% RSLogix 500 project water_filtration_system.RSS, saved by version 8.30.00.16 %
PROJECT "UNTITLED"    % processor: Bul.1763 MicroLogix 1100 Series B %

PROGRAM FILES
  LAD 2   12 rungs
  LAD 3 "IO"  13 rungs
  LAD 4 "ALARMS"  18 rungs
  LAD 5 "CTRL"  8 rungs
  LAD 6 "HOA"  23 rungs
  LAD 7 "SIM"  7 rungs
  LAD 8 "MODE"  4 rungs
  LAD 9 "BACKWASH"  16 rungs
  LAD 10 "LEVEL"  5 rungs
  LAD 11 "HOURMETER"  8 rungs
  LAD 12 "REVIEW"  7 rungs

DATA FILES
  O0 OUTPUT  4 elements
  I1 INPUT  6 elements
  S2 STATUS  66 elements
  B3 BINARY  7 elements
  T4 TIMER  15 elements
  C5 COUNTER  1 elements
  R6 CONTROL  1 elements
  N7 INTEGER  13 elements
  F8 FLOAT  12 elements
  B9 DIGITAL IO  1 elements
  N10 ANALOG IO  3 elements

LADDER 2
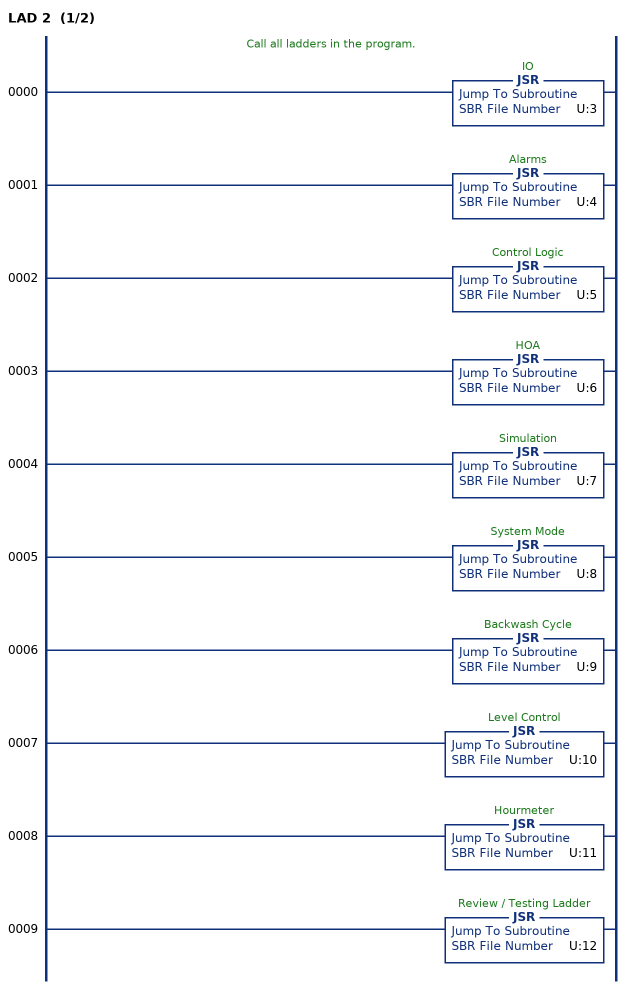
% Rung: 0 %
% Call all ladders in the program. %
SOR JSR U:3 EOR
%   U:3  "IO" %
% Rung: 1 %
SOR JSR U:4 EOR
%   U:4  "Alarms" %
% Rung: 2 %
SOR JSR U:5 EOR
%   U:5  "Control Logic" %
% Rung: 3 %
SOR JSR U:6 EOR
%   U:6  "HOA" %
% Rung: 4 %
SOR JSR U:7 EOR
%   U:7  "Simulation" %
% Rung: 5 %
SOR JSR U:8 EOR
%   U:8  "System Mode" %
% Rung: 6 %
SOR JSR U:9 EOR
%   U:9  "Backwash Cycle" %
% Rung: 7 %
SOR JSR U:10 EOR
%   U:10  "Level Control" %
% Rung: 8 %
SOR JSR U:11 EOR
%   U:11  "Hourmeter" %
% Rung: 9 %
SOR JSR U:12 EOR
%   U:12  "Review / Testing Ladder" %

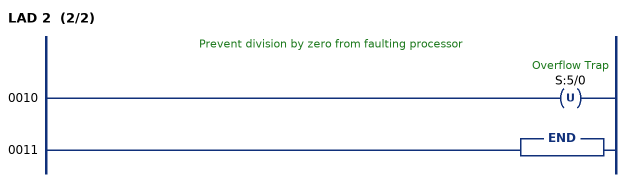
% Rung: 10 %
% Prevent division by zero from faulting processor %
SOR OTU S:5/0 EOR
%   S:5/0  "Overflow Trap" %
% Rung: 11 %
SOR END EOR

LADDER 3 "IO"
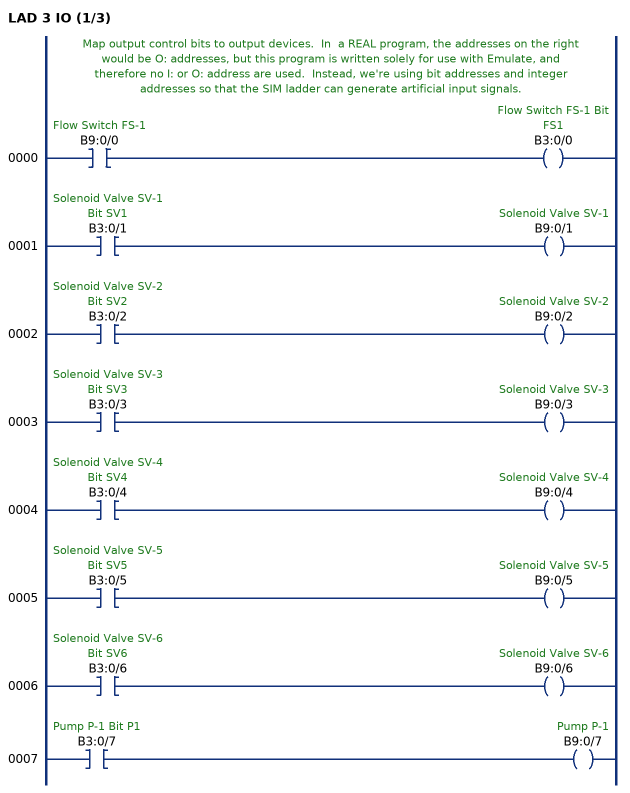
% Rung: 0 %
% Map output control bits to output devices.  In  a REAL program, the addresses on the right would be O: addresses, but this program is written solely for use with Emulate, and therefore no I: or O: address are used.  Instead, we're using bit addresses and integer addresses so that the SIM ladder can generate artificial input signals. %
SOR XIC B9:0/0 OTE B3:0/0 EOR
%   B9:0/0  "Flow Switch FS-1" %
%   B3:0/0  FS1  "Flow Switch FS-1 Bit" %
% Rung: 1 %
SOR XIC B3:0/1 OTE B9:0/1 EOR
%   B3:0/1  SV1  "Solenoid Valve SV-1 Bit" %
%   B9:0/1  "Solenoid Valve SV-1" %
% Rung: 2 %
SOR XIC B3:0/2 OTE B9:0/2 EOR
%   B3:0/2  SV2  "Solenoid Valve SV-2 Bit" %
%   B9:0/2  "Solenoid Valve SV-2" %
% Rung: 3 %
SOR XIC B3:0/3 OTE B9:0/3 EOR
%   B3:0/3  SV3  "Solenoid Valve SV-3 Bit" %
%   B9:0/3  "Solenoid Valve SV-3" %
% Rung: 4 %
SOR XIC B3:0/4 OTE B9:0/4 EOR
%   B3:0/4  SV4  "Solenoid Valve SV-4 Bit" %
%   B9:0/4  "Solenoid Valve SV-4" %
% Rung: 5 %
SOR XIC B3:0/5 OTE B9:0/5 EOR
%   B3:0/5  SV5  "Solenoid Valve SV-5 Bit" %
%   B9:0/5  "Solenoid Valve SV-5" %
% Rung: 6 %
SOR XIC B3:0/6 OTE B9:0/6 EOR
%   B3:0/6  SV6  "Solenoid Valve SV-6 Bit" %
%   B9:0/6  "Solenoid Valve SV-6" %
% Rung: 7 %
SOR XIC B3:0/7 OTE B9:0/7 EOR
%   B3:0/7  P1  "Pump P-1 Bit" %
%   B9:0/7  "Pump P-1" %

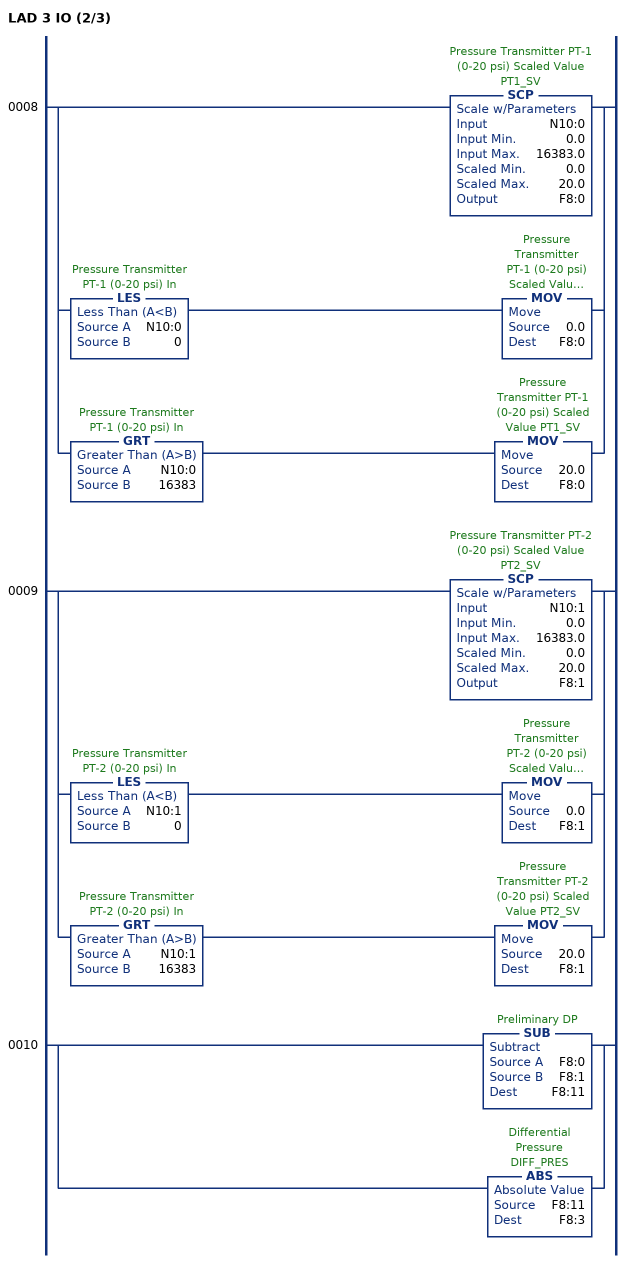
% Rung: 8 %
SOR BST SCP N10:0 0.0 16383.0 0.0 20.0 F8:0 NXB LES N10:0 0 MOV 0.0 F8:0 NXB GRT N10:0 16383 MOV 20.0 F8:0 BND EOR
%   N10:0  "Pressure Transmitter PT-1 (0-20 psi) In" %
%   F8:0  PT1_SV  "Pressure Transmitter PT-1 (0-20 psi) Scaled Value" %
% Rung: 9 %
SOR BST SCP N10:1 0.0 16383.0 0.0 20.0 F8:1 NXB LES N10:1 0 MOV 0.0 F8:1 NXB GRT N10:1 16383 MOV 20.0 F8:1 BND EOR
%   N10:1  "Pressure Transmitter PT-2 (0-20 psi) In" %
%   F8:1  PT2_SV  "Pressure Transmitter PT-2 (0-20 psi) Scaled Value" %
% Rung: 10 %
SOR BST SUB F8:0 F8:1 F8:11 NXB ABS F8:11 F8:3 BND EOR
%   F8:0  PT1_SV  "Pressure Transmitter PT-1 (0-20 psi) Scaled Value" %
%   F8:1  PT2_SV  "Pressure Transmitter PT-2 (0-20 psi) Scaled Value" %
%   F8:11  "Preliminary DP" %
%   F8:3  DIFF_PRES  "Differential Pressure" %

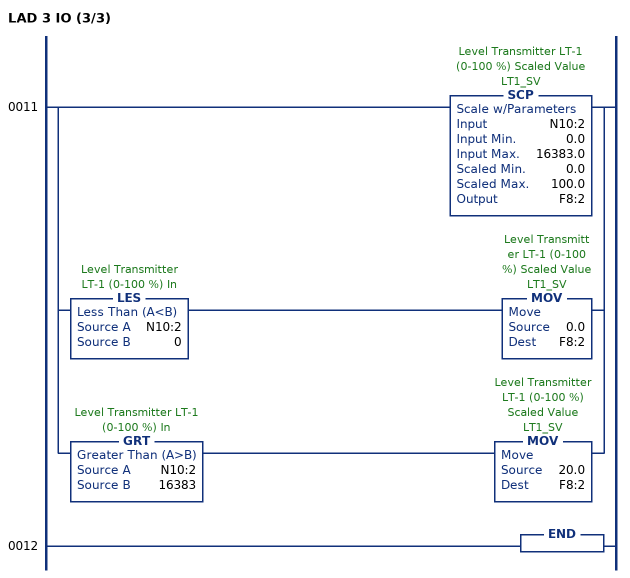
% Rung: 11 %
SOR BST SCP N10:2 0.0 16383.0 0.0 100.0 F8:2 NXB LES N10:2 0 MOV 0.0 F8:2 NXB GRT N10:2 16383 MOV 20.0 F8:2 BND EOR
%   N10:2  "Level Transmitter LT-1 (0-100 %) In" %
%   F8:2  LT1_SV  "Level Transmitter LT-1 (0-100 %) Scaled Value" %
% Rung: 12 %
SOR END EOR

LADDER 4 "ALARMS"
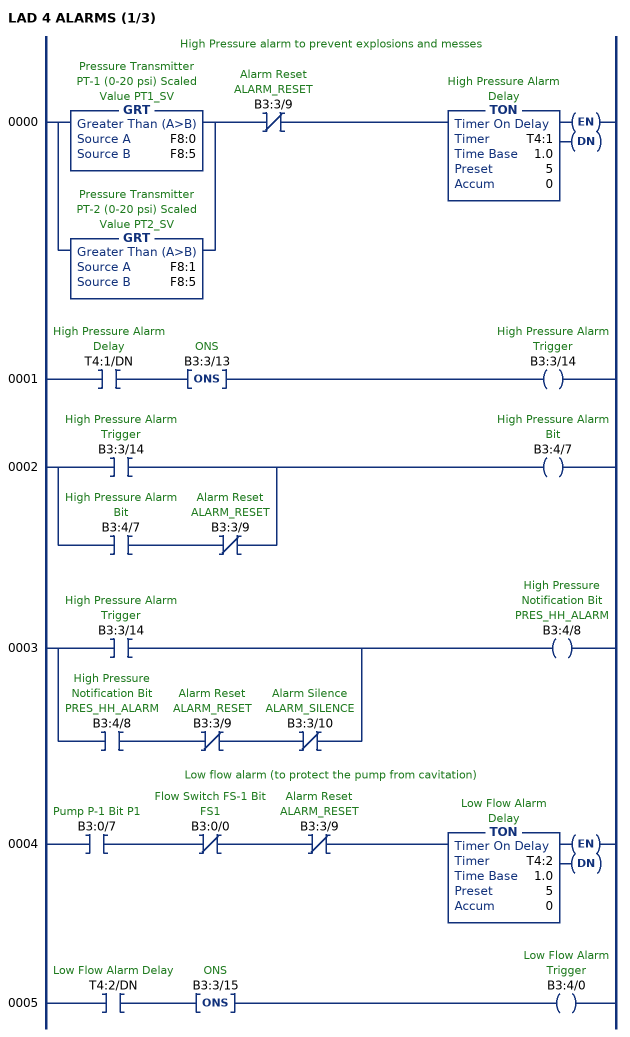
% Rung: 0 %
% High Pressure alarm to prevent explosions and messes %
SOR BST GRT F8:0 F8:5 NXB GRT F8:1 F8:5 BND XIO B3:3/9 TON T4:1 1.0 5 0 EOR
%   F8:0  PT1_SV  "Pressure Transmitter PT-1 (0-20 psi) Scaled Value" %
%   F8:5  PRESSURE_HH_SP  "Pressure HH Alarm Setpoint" %
%   F8:1  PT2_SV  "Pressure Transmitter PT-2 (0-20 psi) Scaled Value" %
%   B3:3/9  ALARM_RESET  "Alarm Reset" %
%   T4:1  "High Pressure Alarm Delay" %
% Rung: 1 %
SOR XIC T4:1/DN ONS B3:3/13 OTE B3:3/14 EOR
%   T4:1  "High Pressure Alarm Delay" %
%   B3:3/13  "ONS" %
%   B3:3/14  "High Pressure Alarm Trigger" %
% Rung: 2 %
SOR BST XIC B3:3/14 NXB XIC B3:4/7 XIO B3:3/9 BND OTE B3:4/7 EOR
%   B3:3/14  "High Pressure Alarm Trigger" %
%   B3:4/7  "High Pressure Alarm Bit" %
%   B3:3/9  ALARM_RESET  "Alarm Reset" %
% Rung: 3 %
SOR BST XIC B3:3/14 NXB XIC B3:4/8 XIO B3:3/9 XIO B3:3/10 BND OTE B3:4/8 EOR
%   B3:3/14  "High Pressure Alarm Trigger" %
%   B3:4/8  PRES_HH_ALARM  "High Pressure Notification Bit" %
%   B3:3/9  ALARM_RESET  "Alarm Reset" %
%   B3:3/10  ALARM_SILENCE  "Alarm Silence" %
% Rung: 4 %
% Low flow alarm (to protect the pump from cavitation) %
SOR XIC B3:0/7 XIO B3:0/0 XIO B3:3/9 TON T4:2 1.0 5 0 EOR
%   B3:0/7  P1  "Pump P-1 Bit" %
%   B3:0/0  FS1  "Flow Switch FS-1 Bit" %
%   B3:3/9  ALARM_RESET  "Alarm Reset" %
%   T4:2  "Low Flow Alarm Delay" %
% Rung: 5 %
SOR XIC T4:2/DN ONS B3:3/15 OTE B3:4/0 EOR
%   T4:2  "Low Flow Alarm Delay" %
%   B3:3/15  "ONS" %
%   B3:4/0  "Low Flow Alarm Trigger" %

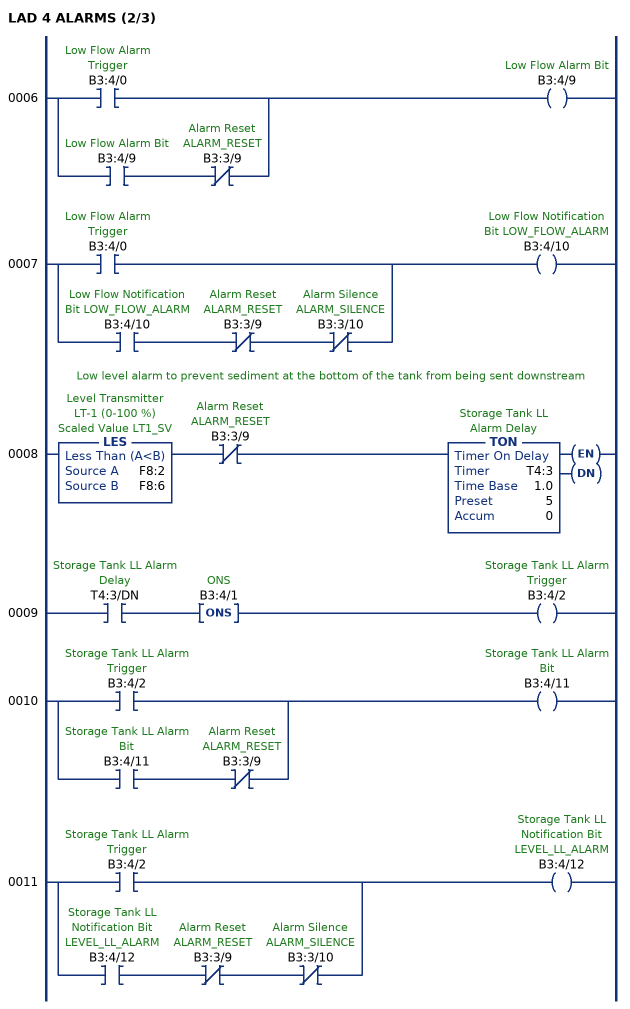
% Rung: 6 %
SOR BST XIC B3:4/0 NXB XIC B3:4/9 XIO B3:3/9 BND OTE B3:4/9 EOR
%   B3:4/0  "Low Flow Alarm Trigger" %
%   B3:4/9  "Low Flow Alarm Bit" %
%   B3:3/9  ALARM_RESET  "Alarm Reset" %
% Rung: 7 %
SOR BST XIC B3:4/0 NXB XIC B3:4/10 XIO B3:3/9 XIO B3:3/10 BND OTE B3:4/10 EOR
%   B3:4/0  "Low Flow Alarm Trigger" %
%   B3:4/10  LOW_FLOW_ALARM  "Low Flow Notification Bit" %
%   B3:3/9  ALARM_RESET  "Alarm Reset" %
%   B3:3/10  ALARM_SILENCE  "Alarm Silence" %
% Rung: 8 %
% Low level alarm to prevent sediment at the bottom of the tank from being sent downstream %
SOR LES F8:2 F8:6 XIO B3:3/9 TON T4:3 1.0 5 0 EOR
%   F8:2  LT1_SV  "Level Transmitter LT-1 (0-100 %) Scaled Value" %
%   F8:6  LEVEL_LL_SP  "Storage Tank LL Alarm Setpoint" %
%   B3:3/9  ALARM_RESET  "Alarm Reset" %
%   T4:3  "Storage Tank LL Alarm Delay" %
% Rung: 9 %
SOR XIC T4:3/DN ONS B3:4/1 OTE B3:4/2 EOR
%   T4:3  "Storage Tank LL Alarm Delay" %
%   B3:4/1  "ONS" %
%   B3:4/2  "Storage Tank LL Alarm Trigger" %
% Rung: 10 %
SOR BST XIC B3:4/2 NXB XIC B3:4/11 XIO B3:3/9 BND OTE B3:4/11 EOR
%   B3:4/2  "Storage Tank LL Alarm Trigger" %
%   B3:4/11  "Storage Tank LL Alarm Bit" %
%   B3:3/9  ALARM_RESET  "Alarm Reset" %
% Rung: 11 %
SOR BST XIC B3:4/2 NXB XIC B3:4/12 XIO B3:3/9 XIO B3:3/10 BND OTE B3:4/12 EOR
%   B3:4/2  "Storage Tank LL Alarm Trigger" %
%   B3:4/12  LEVEL_LL_ALARM  "Storage Tank LL Notification Bit" %
%   B3:3/9  ALARM_RESET  "Alarm Reset" %
%   B3:3/10  ALARM_SILENCE  "Alarm Silence" %

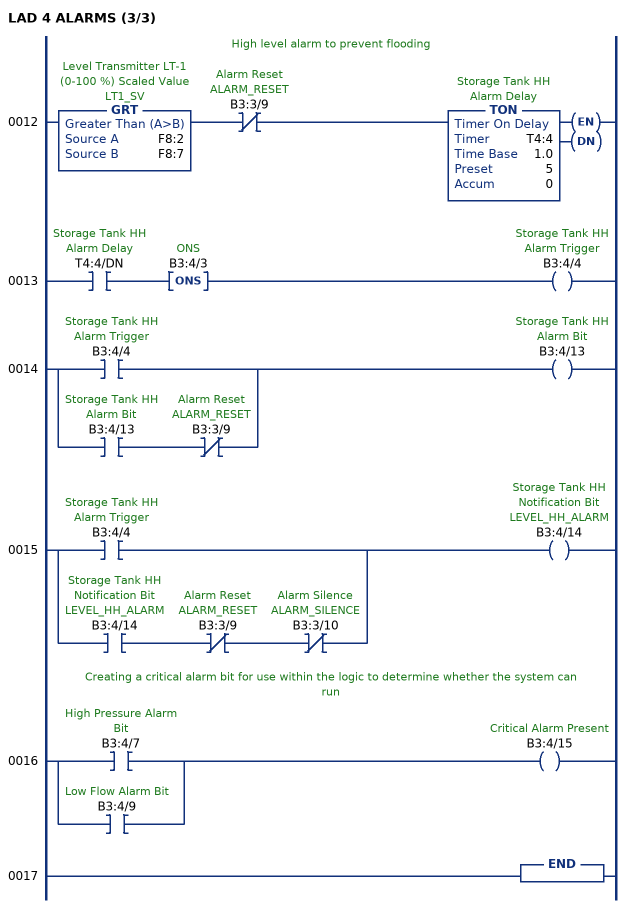
% Rung: 12 %
% High level alarm to prevent flooding %
SOR GRT F8:2 F8:7 XIO B3:3/9 TON T4:4 1.0 5 0 EOR
%   F8:2  LT1_SV  "Level Transmitter LT-1 (0-100 %) Scaled Value" %
%   F8:7  LEVEL_HH_SP  "Storage Tank HH Alarm Setpoint" %
%   B3:3/9  ALARM_RESET  "Alarm Reset" %
%   T4:4  "Storage Tank HH Alarm Delay" %
% Rung: 13 %
SOR XIC T4:4/DN ONS B3:4/3 OTE B3:4/4 EOR
%   T4:4  "Storage Tank HH Alarm Delay" %
%   B3:4/3  "ONS" %
%   B3:4/4  "Storage Tank HH Alarm Trigger" %
% Rung: 14 %
SOR BST XIC B3:4/4 NXB XIC B3:4/13 XIO B3:3/9 BND OTE B3:4/13 EOR
%   B3:4/4  "Storage Tank HH Alarm Trigger" %
%   B3:4/13  "Storage Tank HH Alarm Bit" %
%   B3:3/9  ALARM_RESET  "Alarm Reset" %
% Rung: 15 %
SOR BST XIC B3:4/4 NXB XIC B3:4/14 XIO B3:3/9 XIO B3:3/10 BND OTE B3:4/14 EOR
%   B3:4/4  "Storage Tank HH Alarm Trigger" %
%   B3:4/14  LEVEL_HH_ALARM  "Storage Tank HH Notification Bit" %
%   B3:3/9  ALARM_RESET  "Alarm Reset" %
%   B3:3/10  ALARM_SILENCE  "Alarm Silence" %
% Rung: 16 %
% Creating a critical alarm bit for use within the logic to determine whether the system can run %
SOR BST XIC B3:4/7 NXB XIC B3:4/9 BND OTE B3:4/15 EOR
%   B3:4/7  "High Pressure Alarm Bit" %
%   B3:4/9  "Low Flow Alarm Bit" %
%   B3:4/15  "Critical Alarm Present" %
% Rung: 17 %
SOR END EOR

LADDER 5 "CTRL"
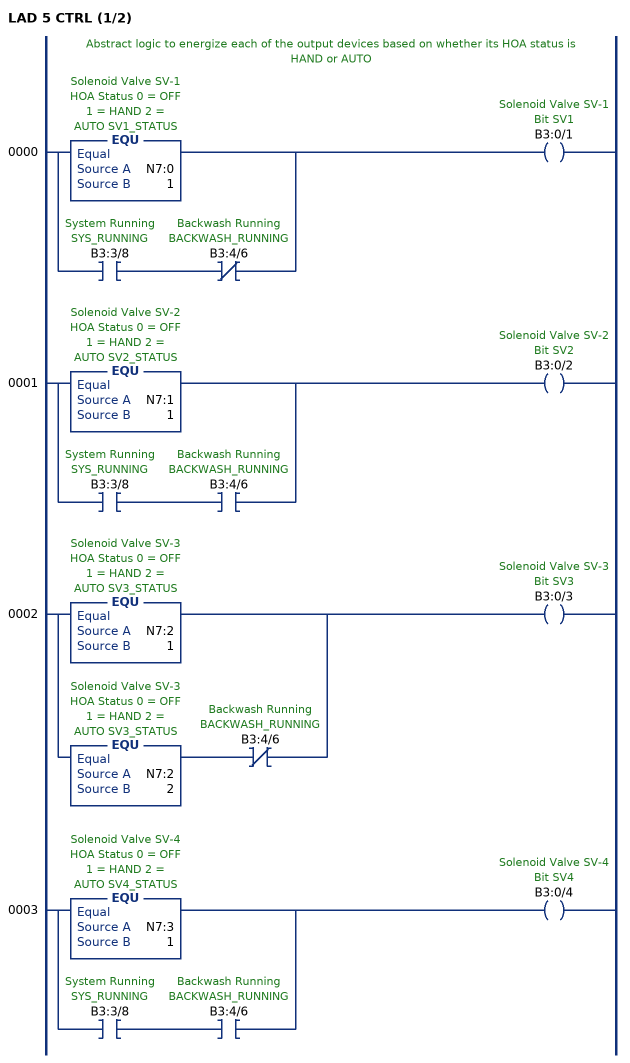
% Rung: 0 %
% Abstract logic to energize each of the output devices based on whether its HOA status is HAND or AUTO %
SOR BST EQU N7:0 1 NXB XIC B3:3/8 XIO B3:4/6 BND OTE B3:0/1 EOR
%   N7:0  SV1_STATUS  "Solenoid Valve SV-1 HOA Status 0 = OFF 1 = HAND 2 = AUTO" %
%   B3:3/8  SYS_RUNNING  "System Running" %
%   B3:4/6  BACKWASH_RUNNING  "Backwash Running" %
%   B3:0/1  SV1  "Solenoid Valve SV-1 Bit" %
% Rung: 1 %
SOR BST EQU N7:1 1 NXB XIC B3:3/8 XIC B3:4/6 BND OTE B3:0/2 EOR
%   N7:1  SV2_STATUS  "Solenoid Valve SV-2 HOA Status 0 = OFF 1 = HAND 2 = AUTO" %
%   B3:3/8  SYS_RUNNING  "System Running" %
%   B3:4/6  BACKWASH_RUNNING  "Backwash Running" %
%   B3:0/2  SV2  "Solenoid Valve SV-2 Bit" %
% Rung: 2 %
SOR BST EQU N7:2 1 NXB EQU N7:2 2 XIO B3:4/6 BND OTE B3:0/3 EOR
%   N7:2  SV3_STATUS  "Solenoid Valve SV-3 HOA Status 0 = OFF 1 = HAND 2 = AUTO" %
%   B3:4/6  BACKWASH_RUNNING  "Backwash Running" %
%   B3:0/3  SV3  "Solenoid Valve SV-3 Bit" %
% Rung: 3 %
SOR BST EQU N7:3 1 NXB XIC B3:3/8 XIC B3:4/6 BND OTE B3:0/4 EOR
%   N7:3  SV4_STATUS  "Solenoid Valve SV-4 HOA Status 0 = OFF 1 = HAND 2 = AUTO" %
%   B3:3/8  SYS_RUNNING  "System Running" %
%   B3:4/6  BACKWASH_RUNNING  "Backwash Running" %
%   B3:0/4  SV4  "Solenoid Valve SV-4 Bit" %

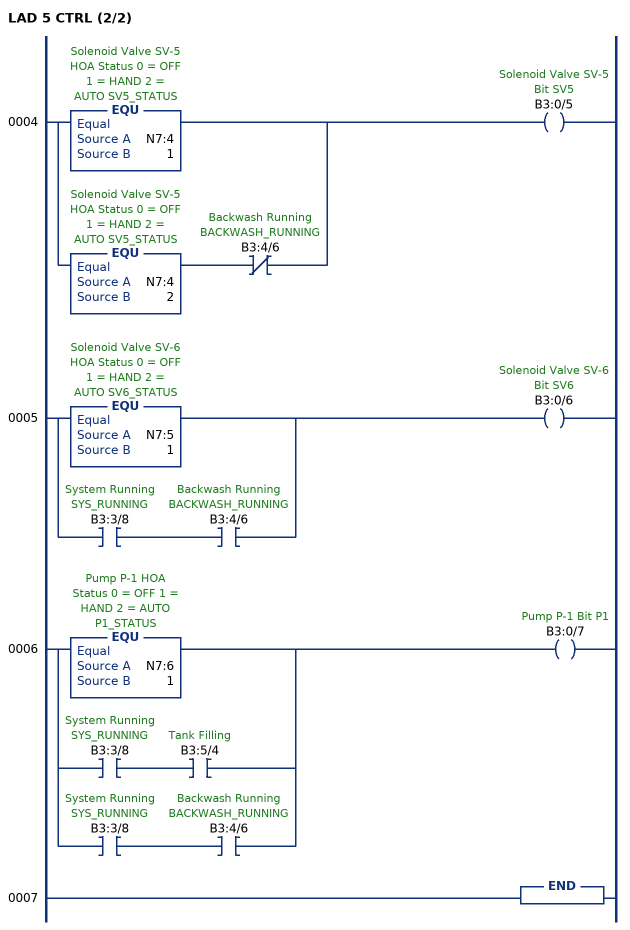
% Rung: 4 %
SOR BST EQU N7:4 1 NXB EQU N7:4 2 XIO B3:4/6 BND OTE B3:0/5 EOR
%   N7:4  SV5_STATUS  "Solenoid Valve SV-5 HOA Status 0 = OFF 1 = HAND 2 = AUTO" %
%   B3:4/6  BACKWASH_RUNNING  "Backwash Running" %
%   B3:0/5  SV5  "Solenoid Valve SV-5 Bit" %
% Rung: 5 %
SOR BST EQU N7:5 1 NXB XIC B3:3/8 XIC B3:4/6 BND OTE B3:0/6 EOR
%   N7:5  SV6_STATUS  "Solenoid Valve SV-6 HOA Status 0 = OFF 1 = HAND 2 = AUTO" %
%   B3:3/8  SYS_RUNNING  "System Running" %
%   B3:4/6  BACKWASH_RUNNING  "Backwash Running" %
%   B3:0/6  SV6  "Solenoid Valve SV-6 Bit" %
% Rung: 6 %
SOR BST EQU N7:6 1 NXB XIC B3:3/8 XIC B3:5/4 NXB XIC B3:3/8 XIC B3:4/6 BND OTE B3:0/7 EOR
%   N7:6  P1_STATUS  "Pump P-1 HOA Status 0 = OFF 1 = HAND 2 = AUTO" %
%   B3:3/8  SYS_RUNNING  "System Running" %
%   B3:5/4  "Tank Filling" %
%   B3:4/6  BACKWASH_RUNNING  "Backwash Running" %
%   B3:0/7  P1  "Pump P-1 Bit" %
% Rung: 7 %
SOR END EOR

LADDER 6 "HOA"
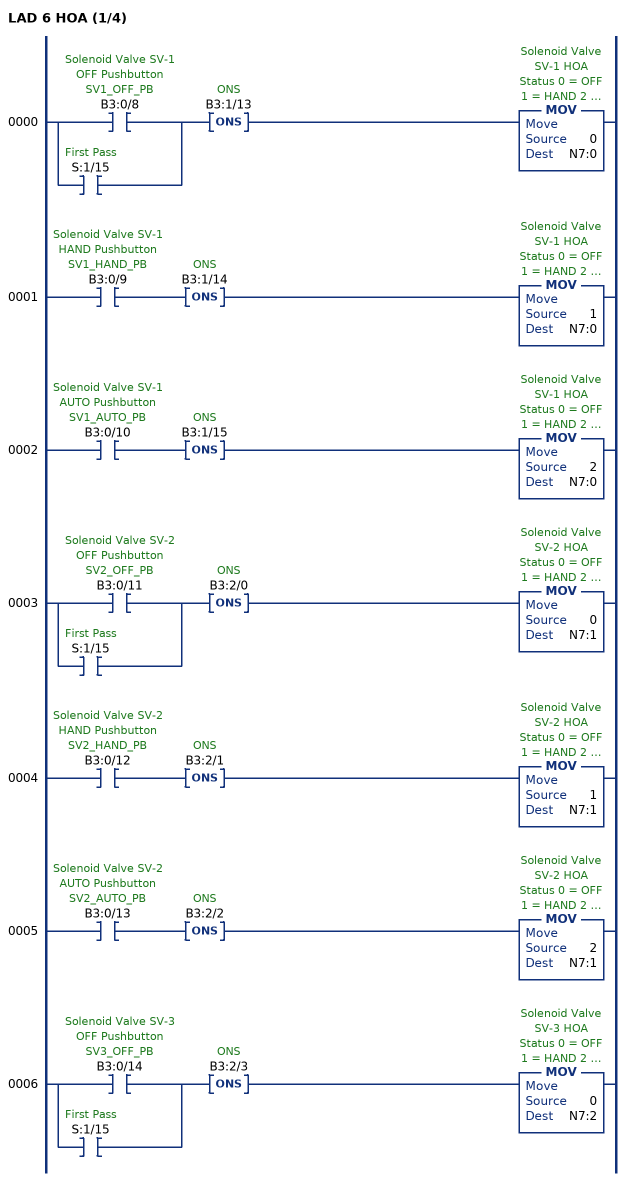
% Rung: 0 %
SOR BST XIC B3:0/8 NXB XIC S:1/15 BND ONS B3:1/13 MOV 0 N7:0 EOR
%   B3:0/8  SV1_OFF_PB  "Solenoid Valve SV-1 OFF Pushbutton" %
%   S:1/15  "First Pass" %
%   B3:1/13  "ONS" %
%   N7:0  SV1_STATUS  "Solenoid Valve SV-1 HOA Status 0 = OFF 1 = HAND 2 = AUTO" %
% Rung: 1 %
SOR XIC B3:0/9 ONS B3:1/14 MOV 1 N7:0 EOR
%   B3:0/9  SV1_HAND_PB  "Solenoid Valve SV-1 HAND Pushbutton" %
%   B3:1/14  "ONS" %
%   N7:0  SV1_STATUS  "Solenoid Valve SV-1 HOA Status 0 = OFF 1 = HAND 2 = AUTO" %
% Rung: 2 %
SOR XIC B3:0/10 ONS B3:1/15 MOV 2 N7:0 EOR
%   B3:0/10  SV1_AUTO_PB  "Solenoid Valve SV-1 AUTO Pushbutton" %
%   B3:1/15  "ONS" %
%   N7:0  SV1_STATUS  "Solenoid Valve SV-1 HOA Status 0 = OFF 1 = HAND 2 = AUTO" %
% Rung: 3 %
SOR BST XIC B3:0/11 NXB XIC S:1/15 BND ONS B3:2/0 MOV 0 N7:1 EOR
%   B3:0/11  SV2_OFF_PB  "Solenoid Valve SV-2 OFF Pushbutton" %
%   S:1/15  "First Pass" %
%   B3:2/0  "ONS" %
%   N7:1  SV2_STATUS  "Solenoid Valve SV-2 HOA Status 0 = OFF 1 = HAND 2 = AUTO" %
% Rung: 4 %
SOR XIC B3:0/12 ONS B3:2/1 MOV 1 N7:1 EOR
%   B3:0/12  SV2_HAND_PB  "Solenoid Valve SV-2 HAND Pushbutton" %
%   B3:2/1  "ONS" %
%   N7:1  SV2_STATUS  "Solenoid Valve SV-2 HOA Status 0 = OFF 1 = HAND 2 = AUTO" %
% Rung: 5 %
SOR XIC B3:0/13 ONS B3:2/2 MOV 2 N7:1 EOR
%   B3:0/13  SV2_AUTO_PB  "Solenoid Valve SV-2 AUTO Pushbutton" %
%   B3:2/2  "ONS" %
%   N7:1  SV2_STATUS  "Solenoid Valve SV-2 HOA Status 0 = OFF 1 = HAND 2 = AUTO" %
% Rung: 6 %
SOR BST XIC B3:0/14 NXB XIC S:1/15 BND ONS B3:2/3 MOV 0 N7:2 EOR
%   B3:0/14  SV3_OFF_PB  "Solenoid Valve SV-3 OFF Pushbutton" %
%   S:1/15  "First Pass" %
%   B3:2/3  "ONS" %
%   N7:2  SV3_STATUS  "Solenoid Valve SV-3 HOA Status 0 = OFF 1 = HAND 2 = AUTO" %

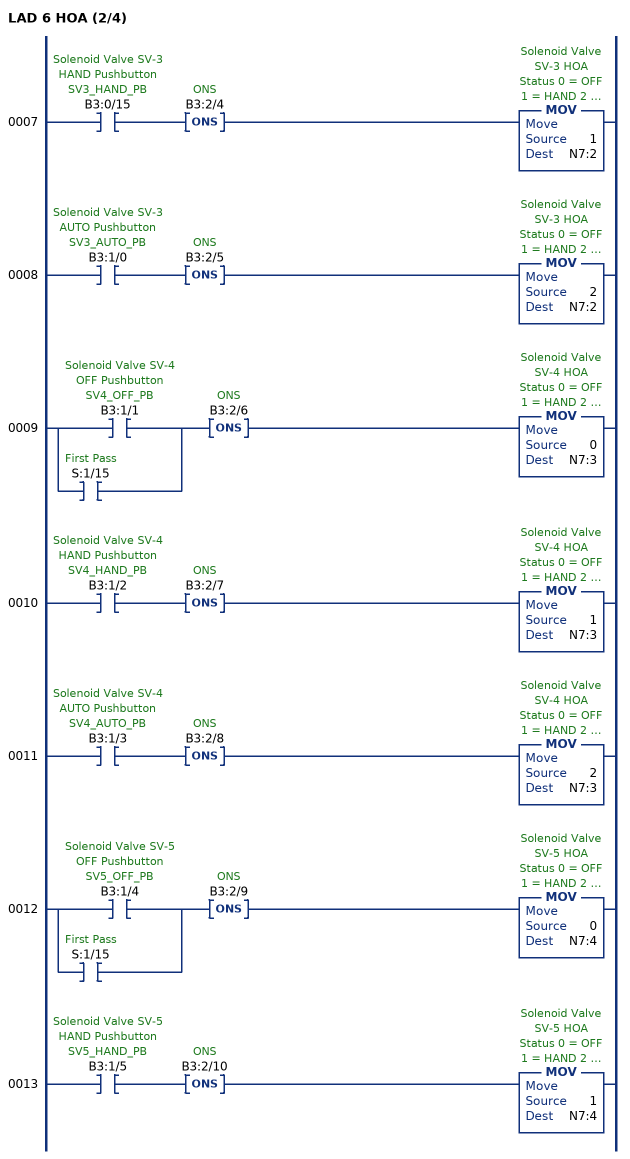
% Rung: 7 %
SOR XIC B3:0/15 ONS B3:2/4 MOV 1 N7:2 EOR
%   B3:0/15  SV3_HAND_PB  "Solenoid Valve SV-3 HAND Pushbutton" %
%   B3:2/4  "ONS" %
%   N7:2  SV3_STATUS  "Solenoid Valve SV-3 HOA Status 0 = OFF 1 = HAND 2 = AUTO" %
% Rung: 8 %
SOR XIC B3:1/0 ONS B3:2/5 MOV 2 N7:2 EOR
%   B3:1/0  SV3_AUTO_PB  "Solenoid Valve SV-3 AUTO Pushbutton" %
%   B3:2/5  "ONS" %
%   N7:2  SV3_STATUS  "Solenoid Valve SV-3 HOA Status 0 = OFF 1 = HAND 2 = AUTO" %
% Rung: 9 %
SOR BST XIC B3:1/1 NXB XIC S:1/15 BND ONS B3:2/6 MOV 0 N7:3 EOR
%   B3:1/1  SV4_OFF_PB  "Solenoid Valve SV-4 OFF Pushbutton" %
%   S:1/15  "First Pass" %
%   B3:2/6  "ONS" %
%   N7:3  SV4_STATUS  "Solenoid Valve SV-4 HOA Status 0 = OFF 1 = HAND 2 = AUTO" %
% Rung: 10 %
SOR XIC B3:1/2 ONS B3:2/7 MOV 1 N7:3 EOR
%   B3:1/2  SV4_HAND_PB  "Solenoid Valve SV-4 HAND Pushbutton" %
%   B3:2/7  "ONS" %
%   N7:3  SV4_STATUS  "Solenoid Valve SV-4 HOA Status 0 = OFF 1 = HAND 2 = AUTO" %
% Rung: 11 %
SOR XIC B3:1/3 ONS B3:2/8 MOV 2 N7:3 EOR
%   B3:1/3  SV4_AUTO_PB  "Solenoid Valve SV-4 AUTO Pushbutton" %
%   B3:2/8  "ONS" %
%   N7:3  SV4_STATUS  "Solenoid Valve SV-4 HOA Status 0 = OFF 1 = HAND 2 = AUTO" %
% Rung: 12 %
SOR BST XIC B3:1/4 NXB XIC S:1/15 BND ONS B3:2/9 MOV 0 N7:4 EOR
%   B3:1/4  SV5_OFF_PB  "Solenoid Valve SV-5 OFF Pushbutton" %
%   S:1/15  "First Pass" %
%   B3:2/9  "ONS" %
%   N7:4  SV5_STATUS  "Solenoid Valve SV-5 HOA Status 0 = OFF 1 = HAND 2 = AUTO" %
% Rung: 13 %
SOR XIC B3:1/5 ONS B3:2/10 MOV 1 N7:4 EOR
%   B3:1/5  SV5_HAND_PB  "Solenoid Valve SV-5 HAND Pushbutton" %
%   B3:2/10  "ONS" %
%   N7:4  SV5_STATUS  "Solenoid Valve SV-5 HOA Status 0 = OFF 1 = HAND 2 = AUTO" %

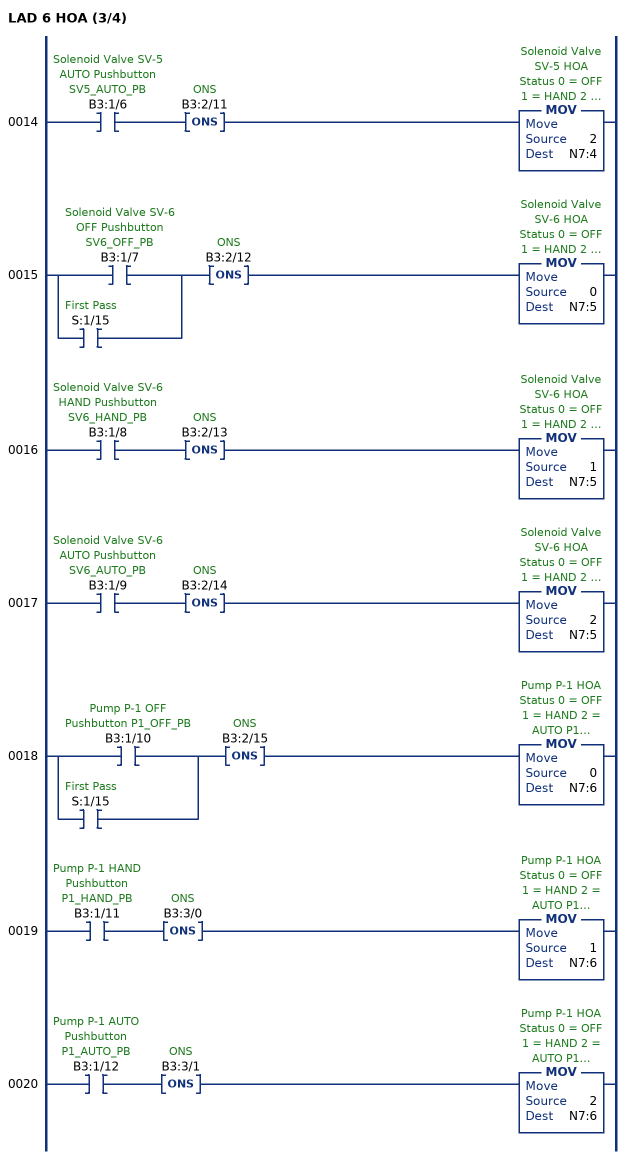
% Rung: 14 %
SOR XIC B3:1/6 ONS B3:2/11 MOV 2 N7:4 EOR
%   B3:1/6  SV5_AUTO_PB  "Solenoid Valve SV-5 AUTO Pushbutton" %
%   B3:2/11  "ONS" %
%   N7:4  SV5_STATUS  "Solenoid Valve SV-5 HOA Status 0 = OFF 1 = HAND 2 = AUTO" %
% Rung: 15 %
SOR BST XIC B3:1/7 NXB XIC S:1/15 BND ONS B3:2/12 MOV 0 N7:5 EOR
%   B3:1/7  SV6_OFF_PB  "Solenoid Valve SV-6 OFF Pushbutton" %
%   S:1/15  "First Pass" %
%   B3:2/12  "ONS" %
%   N7:5  SV6_STATUS  "Solenoid Valve SV-6 HOA Status 0 = OFF 1 = HAND 2 = AUTO" %
% Rung: 16 %
SOR XIC B3:1/8 ONS B3:2/13 MOV 1 N7:5 EOR
%   B3:1/8  SV6_HAND_PB  "Solenoid Valve SV-6 HAND Pushbutton" %
%   B3:2/13  "ONS" %
%   N7:5  SV6_STATUS  "Solenoid Valve SV-6 HOA Status 0 = OFF 1 = HAND 2 = AUTO" %
% Rung: 17 %
SOR XIC B3:1/9 ONS B3:2/14 MOV 2 N7:5 EOR
%   B3:1/9  SV6_AUTO_PB  "Solenoid Valve SV-6 AUTO Pushbutton" %
%   B3:2/14  "ONS" %
%   N7:5  SV6_STATUS  "Solenoid Valve SV-6 HOA Status 0 = OFF 1 = HAND 2 = AUTO" %
% Rung: 18 %
SOR BST XIC B3:1/10 NXB XIC S:1/15 BND ONS B3:2/15 MOV 0 N7:6 EOR
%   B3:1/10  P1_OFF_PB  "Pump P-1 OFF Pushbutton" %
%   S:1/15  "First Pass" %
%   B3:2/15  "ONS" %
%   N7:6  P1_STATUS  "Pump P-1 HOA Status 0 = OFF 1 = HAND 2 = AUTO" %
% Rung: 19 %
SOR XIC B3:1/11 ONS B3:3/0 MOV 1 N7:6 EOR
%   B3:1/11  P1_HAND_PB  "Pump P-1 HAND Pushbutton" %
%   B3:3/0  "ONS" %
%   N7:6  P1_STATUS  "Pump P-1 HOA Status 0 = OFF 1 = HAND 2 = AUTO" %
% Rung: 20 %
SOR XIC B3:1/12 ONS B3:3/1 MOV 2 N7:6 EOR
%   B3:1/12  P1_AUTO_PB  "Pump P-1 AUTO Pushbutton" %
%   B3:3/1  "ONS" %
%   N7:6  P1_STATUS  "Pump P-1 HOA Status 0 = OFF 1 = HAND 2 = AUTO" %

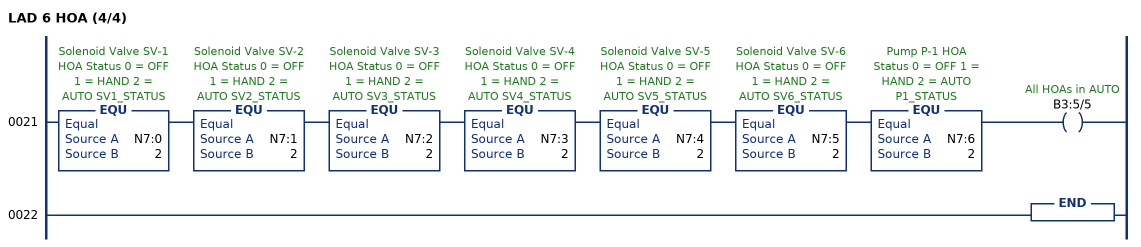
% Rung: 21 %
SOR EQU N7:0 2 EQU N7:1 2 EQU N7:2 2 EQU N7:3 2 EQU N7:4 2 EQU N7:5 2 EQU N7:6 2 OTE B3:5/5 EOR
%   N7:0  SV1_STATUS  "Solenoid Valve SV-1 HOA Status 0 = OFF 1 = HAND 2 = AUTO" %
%   N7:1  SV2_STATUS  "Solenoid Valve SV-2 HOA Status 0 = OFF 1 = HAND 2 = AUTO" %
%   N7:2  SV3_STATUS  "Solenoid Valve SV-3 HOA Status 0 = OFF 1 = HAND 2 = AUTO" %
%   N7:3  SV4_STATUS  "Solenoid Valve SV-4 HOA Status 0 = OFF 1 = HAND 2 = AUTO" %
%   N7:4  SV5_STATUS  "Solenoid Valve SV-5 HOA Status 0 = OFF 1 = HAND 2 = AUTO" %
%   N7:5  SV6_STATUS  "Solenoid Valve SV-6 HOA Status 0 = OFF 1 = HAND 2 = AUTO" %
%   N7:6  P1_STATUS  "Pump P-1 HOA Status 0 = OFF 1 = HAND 2 = AUTO" %
%   B3:5/5  "All HOAs in AUTO" %
% Rung: 22 %
SOR END EOR

LADDER 7 "SIM"
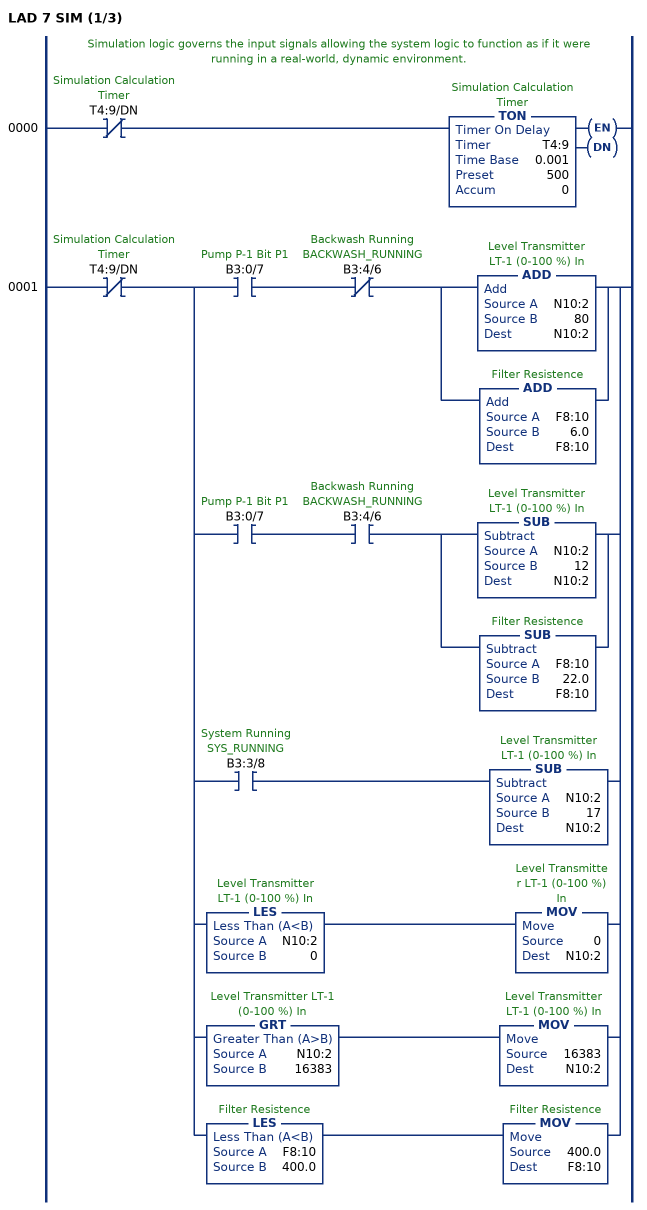
% Rung: 0 %
% Simulation logic governs the input signals allowing the system logic to function as if it were running in a real-world, dynamic environment. %
SOR XIO T4:9/DN TON T4:9 0.001 500 0 EOR
%   T4:9  "Simulation Calculation Timer" %
% Rung: 1 %
SOR XIO T4:9/DN BST XIC B3:0/7 XIO B3:4/6 BST ADD N10:2 80 N10:2 NXB ADD F8:10 6.0 F8:10 BND NXB XIC B3:0/7 XIC B3:4/6 BST SUB N10:2 12 N10:2 NXB SUB F8:10 22.0 F8:10 BND NXB XIC B3:3/8 SUB N10:2 17 N10:2 NXB LES N10:2 0 MOV 0 N10:2 NXB GRT N10:2 16383 MOV 16383 N10:2 NXB LES F8:10 400.0 MOV 400.0 F8:10 BND EOR
%   T4:9  "Simulation Calculation Timer" %
%   B3:0/7  P1  "Pump P-1 Bit" %
%   B3:4/6  BACKWASH_RUNNING  "Backwash Running" %
%   N10:2  "Level Transmitter LT-1 (0-100 %) In" %
%   F8:10  "Filter Resistence" %
%   B3:3/8  SYS_RUNNING  "System Running" %

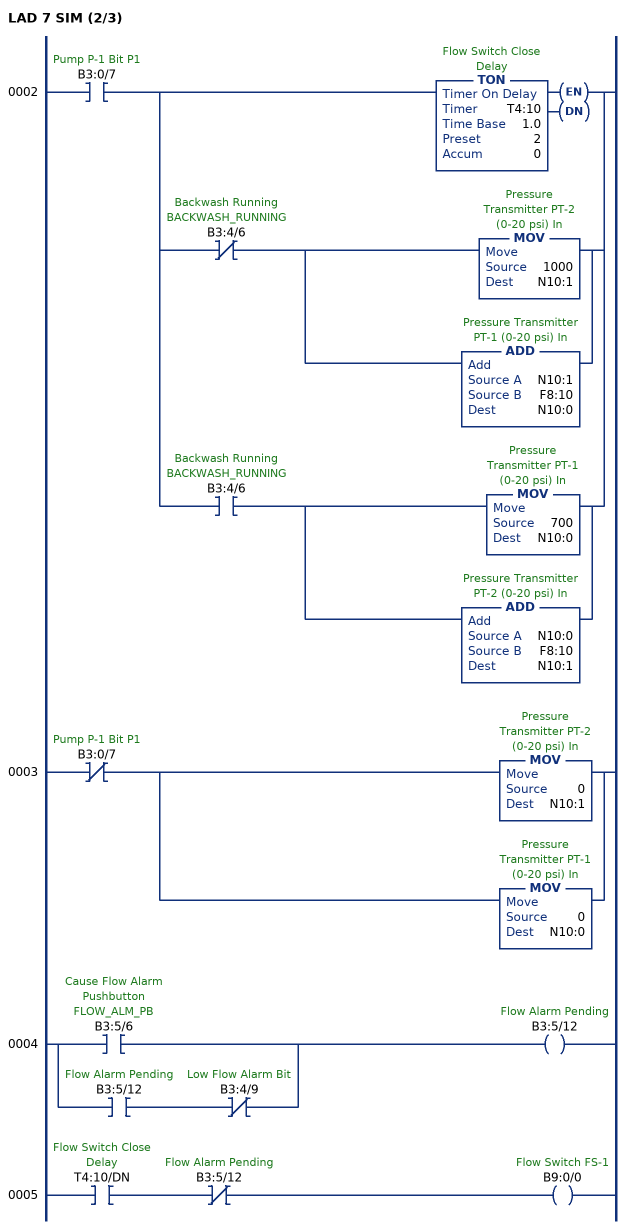
% Rung: 2 %
SOR XIC B3:0/7 BST TON T4:10 1.0 2 0 NXB XIO B3:4/6 BST MOV 1000 N10:1 NXB ADD N10:1 F8:10 N10:0 BND NXB XIC B3:4/6 BST MOV 700 N10:0 NXB ADD N10:0 F8:10 N10:1 BND BND EOR
%   B3:0/7  P1  "Pump P-1 Bit" %
%   T4:10  "Flow Switch Close Delay" %
%   B3:4/6  BACKWASH_RUNNING  "Backwash Running" %
%   N10:1  "Pressure Transmitter PT-2 (0-20 psi) In" %
%   F8:10  "Filter Resistence" %
%   N10:0  "Pressure Transmitter PT-1 (0-20 psi) In" %
% Rung: 3 %
SOR XIO B3:0/7 BST MOV 0 N10:1 NXB MOV 0 N10:0 BND EOR
%   B3:0/7  P1  "Pump P-1 Bit" %
%   N10:1  "Pressure Transmitter PT-2 (0-20 psi) In" %
%   N10:0  "Pressure Transmitter PT-1 (0-20 psi) In" %
% Rung: 4 %
SOR BST XIC B3:5/6 NXB XIC B3:5/12 XIO B3:4/9 BND OTE B3:5/12 EOR
%   B3:5/6  FLOW_ALM_PB  "Cause Flow Alarm Pushbutton" %
%   B3:5/12  "Flow Alarm Pending" %
%   B3:4/9  "Low Flow Alarm Bit" %
% Rung: 5 %
SOR XIC T4:10/DN XIO B3:5/12 OTE B9:0/0 EOR
%   T4:10  "Flow Switch Close Delay" %
%   B3:5/12  "Flow Alarm Pending" %
%   B9:0/0  "Flow Switch FS-1" %

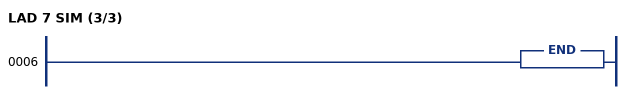
% Rung: 6 %
SOR END EOR

LADDER 8 "MODE"
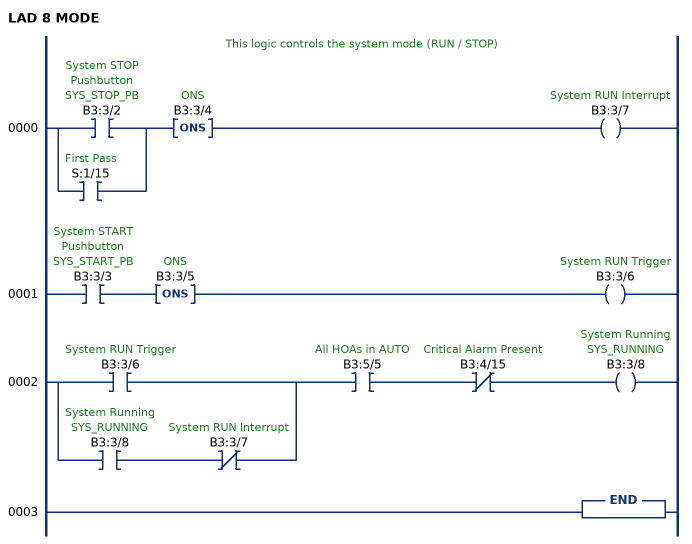
% Rung: 0 %
% This logic controls the system mode (RUN / STOP) %
SOR BST XIC B3:3/2 NXB XIC S:1/15 BND ONS B3:3/4 OTE B3:3/7 EOR
%   B3:3/2  SYS_STOP_PB  "System STOP Pushbutton" %
%   S:1/15  "First Pass" %
%   B3:3/4  "ONS" %
%   B3:3/7  "System RUN Interrupt" %
% Rung: 1 %
SOR XIC B3:3/3 ONS B3:3/5 OTE B3:3/6 EOR
%   B3:3/3  SYS_START_PB  "System START Pushbutton" %
%   B3:3/5  "ONS" %
%   B3:3/6  "System RUN Trigger" %
% Rung: 2 %
SOR BST XIC B3:3/6 NXB XIC B3:3/8 XIO B3:3/7 BND XIC B3:5/5 XIO B3:4/15 OTE B3:3/8 EOR
%   B3:3/6  "System RUN Trigger" %
%   B3:3/8  SYS_RUNNING  "System Running" %
%   B3:3/7  "System RUN Interrupt" %
%   B3:5/5  "All HOAs in AUTO" %
%   B3:4/15  "Critical Alarm Present" %
% Rung: 3 %
SOR END EOR

LADDER 9 "BACKWASH"
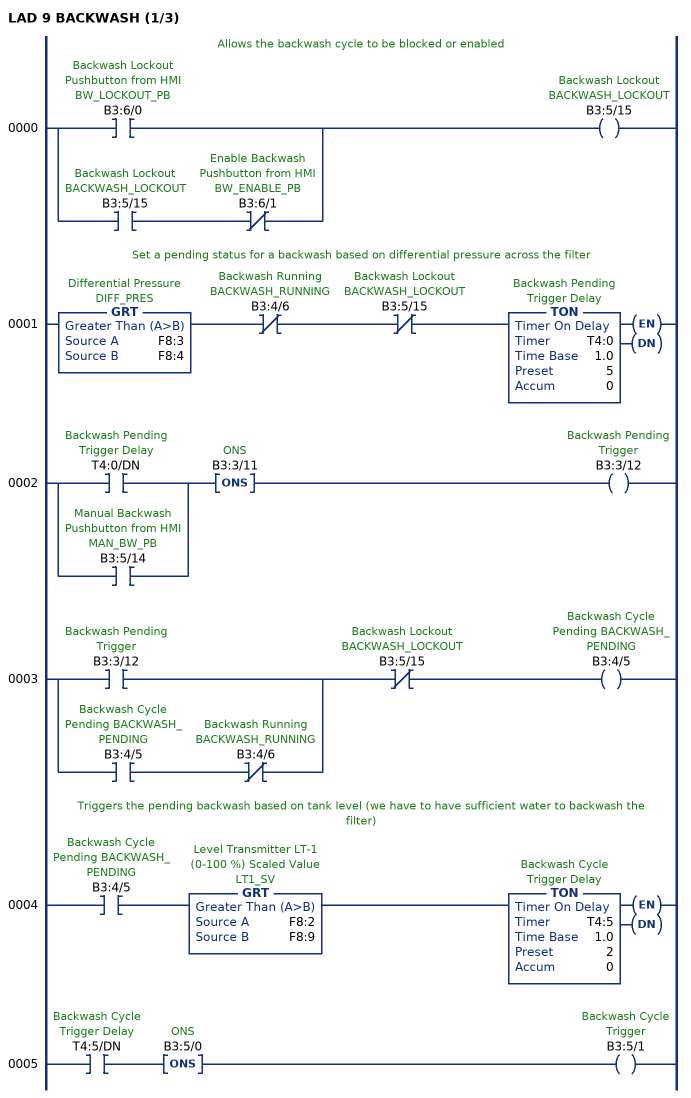
% Rung: 0 %
% Allows the backwash cycle to be blocked or enabled %
SOR BST XIC B3:6/0 NXB XIC B3:5/15 XIO B3:6/1 BND OTE B3:5/15 EOR
%   B3:6/0  BW_LOCKOUT_PB  "Backwash Lockout Pushbutton from HMI" %
%   B3:5/15  BACKWASH_LOCKOUT  "Backwash Lockout" %
%   B3:6/1  BW_ENABLE_PB  "Enable Backwash Pushbutton from HMI" %
% Rung: 1 %
% Set a pending status for a backwash based on differential pressure across the filter %
SOR GRT F8:3 F8:4 XIO B3:4/6 XIO B3:5/15 TON T4:0 1.0 5 0 EOR
%   F8:3  DIFF_PRES  "Differential Pressure" %
%   F8:4  BACKWASH_SP  "Backwash Cycle Trigger Setpoint" %
%   B3:4/6  BACKWASH_RUNNING  "Backwash Running" %
%   B3:5/15  BACKWASH_LOCKOUT  "Backwash Lockout" %
%   T4:0  "Backwash Pending Trigger Delay" %
% Rung: 2 %
SOR BST XIC T4:0/DN NXB XIC B3:5/14 BND ONS B3:3/11 OTE B3:3/12 EOR
%   T4:0  "Backwash Pending Trigger Delay" %
%   B3:5/14  MAN_BW_PB  "Manual Backwash Pushbutton from HMI" %
%   B3:3/11  "ONS" %
%   B3:3/12  "Backwash Pending Trigger" %
% Rung: 3 %
SOR BST XIC B3:3/12 NXB XIC B3:4/5 XIO B3:4/6 BND XIO B3:5/15 OTE B3:4/5 EOR
%   B3:3/12  "Backwash Pending Trigger" %
%   B3:4/5  BACKWASH_PENDING  "Backwash Cycle Pending" %
%   B3:4/6  BACKWASH_RUNNING  "Backwash Running" %
%   B3:5/15  BACKWASH_LOCKOUT  "Backwash Lockout" %
% Rung: 4 %
% Triggers the pending backwash based on tank level (we have to have sufficient water to backwash the filter) %
SOR XIC B3:4/5 GRT F8:2 F8:9 TON T4:5 1.0 2 0 EOR
%   B3:4/5  BACKWASH_PENDING  "Backwash Cycle Pending" %
%   F8:2  LT1_SV  "Level Transmitter LT-1 (0-100 %) Scaled Value" %
%   F8:9  LEVEL_H_SP  "Storage Tank High Level Setpoint" %
%   T4:5  "Backwash Cycle Trigger Delay" %
% Rung: 5 %
SOR XIC T4:5/DN ONS B3:5/0 OTE B3:5/1 EOR
%   T4:5  "Backwash Cycle Trigger Delay" %
%   B3:5/0  "ONS" %
%   B3:5/1  "Backwash Cycle Trigger" %

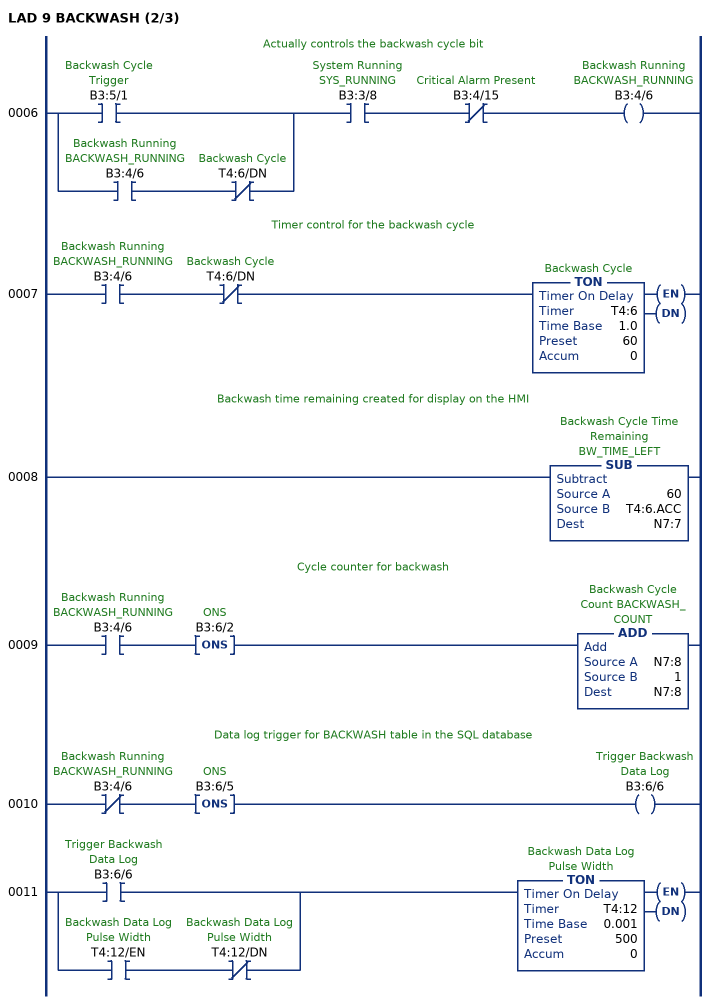
% Rung: 6 %
% Actually controls the backwash cycle bit %
SOR BST XIC B3:5/1 NXB XIC B3:4/6 XIO T4:6/DN BND XIC B3:3/8 XIO B3:4/15 OTE B3:4/6 EOR
%   B3:5/1  "Backwash Cycle Trigger" %
%   B3:4/6  BACKWASH_RUNNING  "Backwash Running" %
%   T4:6  "Backwash Cycle" %
%   B3:3/8  SYS_RUNNING  "System Running" %
%   B3:4/15  "Critical Alarm Present" %
% Rung: 7 %
% Timer control for the backwash cycle %
SOR XIC B3:4/6 XIO T4:6/DN TON T4:6 1.0 60 0 EOR
%   B3:4/6  BACKWASH_RUNNING  "Backwash Running" %
%   T4:6  "Backwash Cycle" %
% Rung: 8 %
% Backwash time remaining created for display on the HMI %
SOR SUB 60 T4:6.ACC N7:7 EOR
%   T4:6  "Backwash Cycle" %
%   N7:7  BW_TIME_LEFT  "Backwash Cycle Time Remaining" %
% Rung: 9 %
% Cycle counter for backwash %
SOR XIC B3:4/6 ONS B3:6/2 ADD N7:8 1 N7:8 EOR
%   B3:4/6  BACKWASH_RUNNING  "Backwash Running" %
%   B3:6/2  "ONS" %
%   N7:8  BACKWASH_COUNT  "Backwash Cycle Count" %
% Rung: 10 %
% Data log trigger for BACKWASH table in the SQL database %
SOR XIO B3:4/6 ONS B3:6/5 OTE B3:6/6 EOR
%   B3:4/6  BACKWASH_RUNNING  "Backwash Running" %
%   B3:6/5  "ONS" %
%   B3:6/6  "Trigger Backwash Data Log" %
% Rung: 11 %
SOR BST XIC B3:6/6 NXB XIC T4:12/EN XIO T4:12/DN BND TON T4:12 0.001 500 0 EOR
%   B3:6/6  "Trigger Backwash Data Log" %
%   T4:12  "Backwash Data Log Pulse Width" %

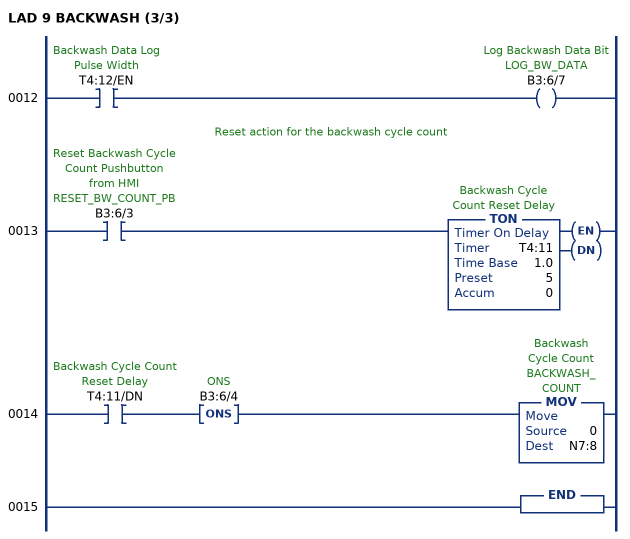
% Rung: 12 %
SOR XIC T4:12/EN OTE B3:6/7 EOR
%   T4:12  "Backwash Data Log Pulse Width" %
%   B3:6/7  LOG_BW_DATA  "Log Backwash Data Bit" %
% Rung: 13 %
% Reset action for the backwash cycle count %
SOR XIC B3:6/3 TON T4:11 1.0 5 0 EOR
%   B3:6/3  RESET_BW_COUNT_PB  "Reset Backwash Cycle Count Pushbutton from HMI" %
%   T4:11  "Backwash Cycle Count Reset Delay" %
% Rung: 14 %
SOR XIC T4:11/DN ONS B3:6/4 MOV 0 N7:8 EOR
%   T4:11  "Backwash Cycle Count Reset Delay" %
%   B3:6/4  "ONS" %
%   N7:8  BACKWASH_COUNT  "Backwash Cycle Count" %
% Rung: 15 %
SOR END EOR

LADDER 10 "LEVEL"
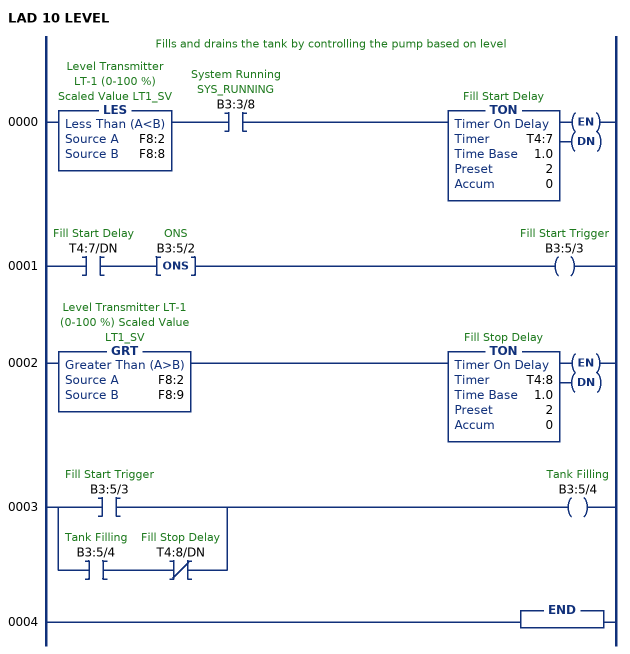
% Rung: 0 %
% Fills and drains the tank by controlling the pump based on level %
SOR LES F8:2 F8:8 XIC B3:3/8 TON T4:7 1.0 2 0 EOR
%   F8:2  LT1_SV  "Level Transmitter LT-1 (0-100 %) Scaled Value" %
%   F8:8  LEVEL_L_SP  "Storage Tank Low Level Setpoint" %
%   B3:3/8  SYS_RUNNING  "System Running" %
%   T4:7  "Fill Start Delay" %
% Rung: 1 %
SOR XIC T4:7/DN ONS B3:5/2 OTE B3:5/3 EOR
%   T4:7  "Fill Start Delay" %
%   B3:5/2  "ONS" %
%   B3:5/3  "Fill Start Trigger" %
% Rung: 2 %
SOR GRT F8:2 F8:9 TON T4:8 1.0 2 0 EOR
%   F8:2  LT1_SV  "Level Transmitter LT-1 (0-100 %) Scaled Value" %
%   F8:9  LEVEL_H_SP  "Storage Tank High Level Setpoint" %
%   T4:8  "Fill Stop Delay" %
% Rung: 3 %
SOR BST XIC B3:5/3 NXB XIC B3:5/4 XIO T4:8/DN BND OTE B3:5/4 EOR
%   B3:5/3  "Fill Start Trigger" %
%   B3:5/4  "Tank Filling" %
%   T4:8  "Fill Stop Delay" %
% Rung: 4 %
SOR END EOR

LADDER 11 "HOURMETER"
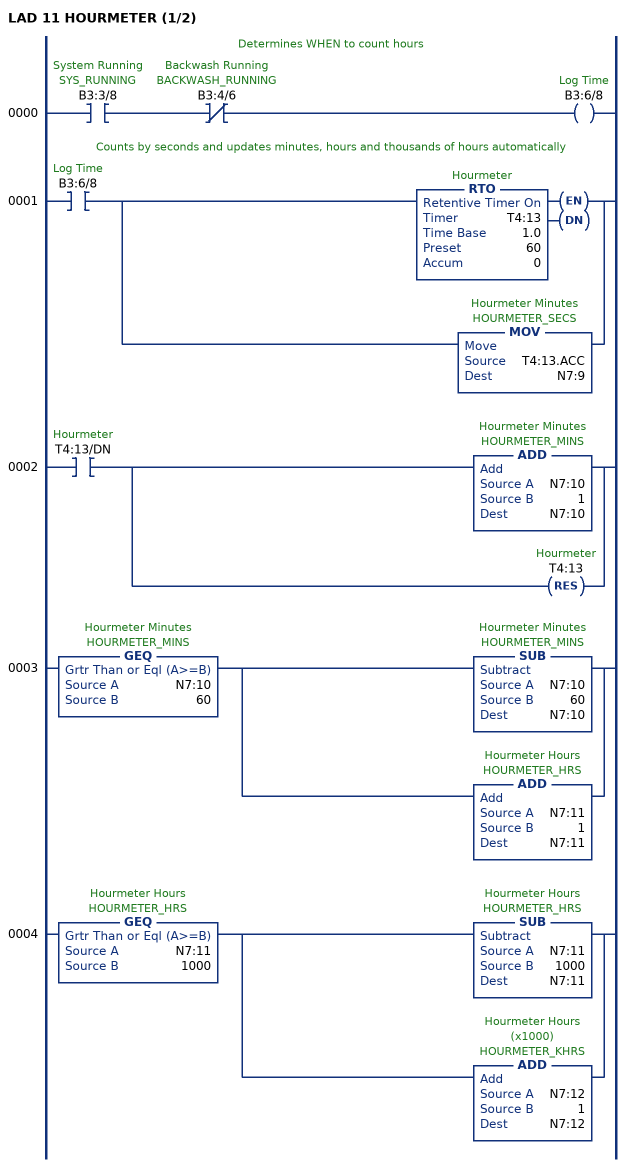
% Rung: 0 %
% Determines WHEN to count hours %
SOR XIC B3:3/8 XIO B3:4/6 OTE B3:6/8 EOR
%   B3:3/8  SYS_RUNNING  "System Running" %
%   B3:4/6  BACKWASH_RUNNING  "Backwash Running" %
%   B3:6/8  "Log Time" %
% Rung: 1 %
% Counts by seconds and updates minutes, hours and thousands of hours automatically %
SOR XIC B3:6/8 BST RTO T4:13 1.0 60 0 NXB MOV T4:13.ACC N7:9 BND EOR
%   B3:6/8  "Log Time" %
%   T4:13  "Hourmeter" %
%   N7:9  HOURMETER_SECS  "Hourmeter Minutes" %
% Rung: 2 %
SOR XIC T4:13/DN BST ADD N7:10 1 N7:10 NXB RES T4:13 BND EOR
%   T4:13  "Hourmeter" %
%   N7:10  HOURMETER_MINS  "Hourmeter Minutes" %
% Rung: 3 %
SOR GEQ N7:10 60 BST SUB N7:10 60 N7:10 NXB ADD N7:11 1 N7:11 BND EOR
%   N7:10  HOURMETER_MINS  "Hourmeter Minutes" %
%   N7:11  HOURMETER_HRS  "Hourmeter Hours" %
% Rung: 4 %
SOR GEQ N7:11 1000 BST SUB N7:11 1000 N7:11 NXB ADD N7:12 1 N7:12 BND EOR
%   N7:11  HOURMETER_HRS  "Hourmeter Hours" %
%   N7:12  HOURMETER_KHRS  "Hourmeter Hours (x1000)" %

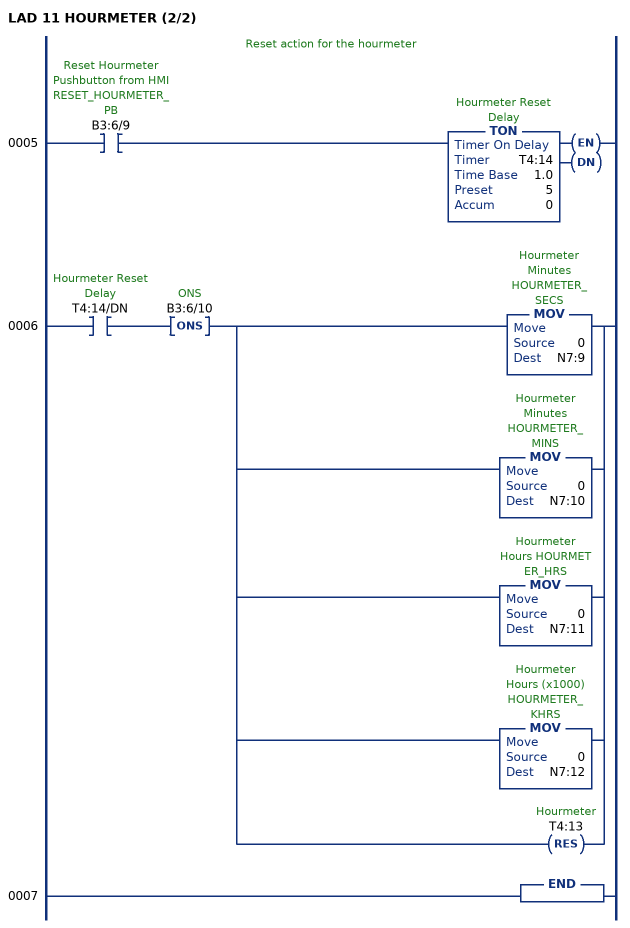
% Rung: 5 %
% Reset action for the hourmeter %
SOR XIC B3:6/9 TON T4:14 1.0 5 0 EOR
%   B3:6/9  RESET_HOURMETER_PB  "Reset Hourmeter Pushbutton from HMI" %
%   T4:14  "Hourmeter Reset Delay" %
% Rung: 6 %
SOR XIC T4:14/DN ONS B3:6/10 BST MOV 0 N7:9 NXB MOV 0 N7:10 NXB MOV 0 N7:11 NXB MOV 0 N7:12 NXB RES T4:13 BND EOR
%   T4:14  "Hourmeter Reset Delay" %
%   B3:6/10  "ONS" %
%   N7:9  HOURMETER_SECS  "Hourmeter Minutes" %
%   N7:10  HOURMETER_MINS  "Hourmeter Minutes" %
%   N7:11  HOURMETER_HRS  "Hourmeter Hours" %
%   N7:12  HOURMETER_KHRS  "Hourmeter Hours (x1000)" %
%   T4:13  "Hourmeter" %
% Rung: 7 %
SOR END EOR

LADDER 12 "REVIEW"
